// TIA Portal V17 export
// export: Created 2023-12-05T13:40:23.7243173Z, ExportSetting WithDefaults, DisplayName Totally Integrated Automation Portal, DisplayVersion V17, DisplayName TIA Portal Openness, DisplayVersion V17, DisplayName TIA Portal Version Control Interface, DisplayVersion V17, DisplayName SINAMICS Startdrive Advanced, DisplayVersion V17, DisplayName SINAMICS Startdrive G130, G150, S120, S150, SINAMICS MV, S210, DisplayVersion V17, DisplayName SINAMICS Startdrive G110M, G120, G120C, G120D, G120P, G115D, DisplayVersion V17, DisplayName STEP 7 Professional, DisplayVersion V17, DisplayName STEP 7 Safety, DisplayVersion V17, DisplayName WinCC Professional, DisplayVersion V17
FUNCTION "KNIFE_COUNTER" : Void   // FC408, LAD
{ S7_Optimized_Access := 'TRUE' }
VERSION : 0.1
// stored: AutoNumber false, IsIECCheckEnabled false, SetENOAutomatically false, UDAEnableTagReadback false
   VAR_INPUT
      Increment_bit : Bool;
      Reset_bit : Bool;
   END_VAR
   VAR_IN_OUT
      CountDOWN : DInt;
      value : DInt;
      Work_Bit1 : Bool;
      Work_Bit2 : Bool;
   END_VAR
BEGIN

NETWORK
TITLE = 
      A     #Increment_bit;
      FP    #Work_Bit1;
      JC    cnt;


      A     #Reset_bit;
      FP    #Work_Bit2;
      JC    rset;
      BEU;

cnt:  L     #CountDOWN;  //LOAD COUNTER DOUBLE DATA WORD
      L     1;
      -D;  //SUB 1 TO DOUBLE DATA WORD
      T     #CountDOWN;  //TRANSFER RESULT BACK TO COUNTER DBD
      BEU;


rset: L     #value;
      T     #CountDOWN;



END_FUNCTION
